Fanuc KAREL source: kb00012.KL

-- PROVISIONAL review KL for V940-1; original PC SHA256 e600cc7b8e4fbd01f44e36c354bb36064a1767b01e4fb5f5dff433a1385a2dec
-- Incomplete behavior may be omitted. Consult companion uncertainty JSON. Do not deploy.
PROGRAM KB00012
%NOLOCKGROUP
BEGIN
  -- V9_ZERO_TABLE_METADATA_HINT layout=0002_ascii; no indexed target words; source/name/runtime held
  -- UNRESOLVED_PC offsets 5-12; opcodes 9D,23
  -- UNRESOLVED_PC offsets 17-24; opcodes 9D,23
  -- UNRESOLVED_PC offsets 29-36; opcodes 9D,23
  -- UNRESOLVED_PC offsets 41-63; opcodes 27,22,22,22,31
  -- UNRESOLVED_PC offsets 68-72; opcodes 7F
END KB00012
